TEXTLIST TL_E_MESSAGETYPE
  0 = 'eMessageEmpty'
  1 = 'eMessageError'
  2 = 'eMessageWarning'
  3 = 'eMessageInfo'
  4 = 'eMessageVerbose'
   = ''
END_TEXTLIST

(* stored: Version 1.1.0.1, ProductVersion 3.1.4026.20
   TextList TL_E_MESSAGETYPE: Id {aa31312a-00ed-4ebd-9139-ba91bc526a12} *)
